(* PLC project cam_computation, Dassault Systèmes ControlBuild 2024x *)
(* stored: creationDateTime 2023-10-04T11:03:50-01:00 *)

(* This module simulates the behavior of a cam profile running module *)
FUNCTION_BLOCK motion_lib.cam_computation
  VAR_INPUT
    profileNr : DINT := 0;
    MasterPositionIn : REAL := 0.0;
  END_VAR
  VAR_INPUT
    nbPoints0 : INT := 0;
    MasterPoints0 : ARRAY[1..100] OF REAL := [100(0.0)];
    SlavePoints0 : ARRAY[1..100] OF REAL := [100(0.0)];
    pointer0 : DINT := 0;
  END_VAR
  VAR_INPUT
    nbPoints1 : INT := 0;
    MasterPoints1 : ARRAY[1..100] OF REAL := [100(0.0)];
    SlavePoints1 : ARRAY[1..100] OF REAL := [100(0.0)];
    pointer1 : DINT := 0;
  END_VAR
  VAR_INPUT
    nbPoints2 : INT := 0;
    MasterPoints2 : ARRAY[1..100] OF REAL := [100(0.0)];
    SlavePoints2 : ARRAY[1..100] OF REAL := [100(0.0)];
    pointer2 : DINT := 0;
  END_VAR
  VAR_INPUT
    nbPoints3 : INT := 0;
    MasterPoints3 : ARRAY[1..100] OF REAL := [100(0.0)];
    SlavePoints3 : ARRAY[1..100] OF REAL := [100(0.0)];
    pointer3 : DINT := 0;
  END_VAR
  VAR_OUTPUT
    slavePosition : REAL := 0.0;
    masterPosition : REAL := 0.0;
  END_VAR
  VAR
    i : INT := 0;
    modulo : REAL := 0.0;
    divider : INT := 0;
    faultProfileNr : BOOL := false;
    faultMasterPositionOOB : BOOL := false;
    faultLinComputation : BOOL := false;
    nbPoints : INT := 0;
    MasterPoints : ARRAY[1..100] OF REAL := [100(0.0)];
    SlavePoints : ARRAY[1..100] OF REAL := [100(0.0)];
    found : BOOL := false;
    index : INT := 0;
    linDenom : REAL := 0.0;
    linNum : REAL := 0.0;
    linA : REAL := 0.0;
    linB : REAL := 0.0;
  END_VAR
  VAR CONSTANT
    FACTOR : REAL := 1.0;
  END_VAR


ACTION C_source_code:
/* ----------------------------------------------------------------	*/
/* Type : Model of Operative Behaviour					*/
/* Category : motion_control						*/
/* Author : Dassault Systemes						*/
/* Update date : June 2021							*/
/* ----------------------------------------------------------------	*/
/* This module do the Slave cam computation from one Master position	*/
/* The profile table inputs are provided by the module cam_profile	*/
/* It's possible to switch in real time between 4 different profiles	*/
/* ----------------------------------------------------------------	*/


if (profileNr<0 || profileNr>3) {
	faultProfileNr = 1;
} else {
	faultProfileNr = 0;
	if (profileNr==0 && nbPoints0) {
		camTable = pointer0;
		nbPoints = nbPoints0;
		for (i=1; i< 100; i++) {
			MasterPoints(i) = camTable->master[i-1];
			SlavePoints(i) = camTable->slave[i-1];
		}
		modulo = camTable->master[nbPoints-1];
	} else {
		if (profileNr==1 && nbPoints1) {
			camTable = pointer1;
			nbPoints = nbPoints1;
			for (i=1; i< 100; i++) {
				MasterPoints(i) = camTable->master[i-1];
				SlavePoints(i) = camTable->slave[i-1];
			}
			modulo = camTable->master[nbPoints-1];
		} else {
			if (profileNr==2 && nbPoints2) {
				camTable = pointer2;
				nbPoints = nbPoints2;
				for (i=1; i< 100; i++) {
					MasterPoints(i) = camTable->master[i-1];
					SlavePoints(i) = camTable->slave[i-1];
				}
				modulo = camTable->master[nbPoints-1];
			} else {
				if (profileNr==3 && nbPoints3) {
					camTable = pointer3;
					nbPoints = nbPoints3;
					for (i=1; i< 100; i++) {
						MasterPoints(i) = camTable->master[i-1];
						SlavePoints(i) = camTable->slave[i-1];
					}
					modulo = camTable->master[nbPoints-1];
				}
			}
		}
	}
	if (nbPoints >= 2) {
		masterPosition = MasterPositionIn - divider * modulo;
		while (masterPosition > modulo) {
			divider += 1;
			masterPosition = MasterPositionIn - divider * modulo;
		}
		while (masterPosition < 0) {
			divider -= 1;
			masterPosition = MasterPositionIn - divider * modulo;
		}
		found = 0;
		for (i=1; i<= nbPoints - 1 && found == 0; i++) {
			if (camTable->master[i-1] <= masterPosition && masterPosition <= camTable->master[i]) {
				index = i;
				found = 1;
			} 
		}
		if (!found) {
			faultMasterPositionOOB = 1;
			if (masterPosition < camTable->master[0]) {
				slavePosition = camTable->slave[0] * FACTOR;
			} else {
				slavePosition = SlavePoints(nbPoints) * FACTOR;
			}
		} else {
			linDenom = camTable->master[index] - camTable->master[index-1];
			if (linDenom != 0.0) {
				faultLinComputation = 0;
				linNum = camTable->slave[index] - camTable->slave[index-1];
				linA = linNum / linDenom;
				linB = camTable->slave[index-1] - (linA * camTable->master[index-1]);
				slavePosition = FACTOR * (linA * masterPosition + linB);
			} else {
				faultLinComputation = 1;
			}
		}
	} else {
		slavePosition = 0;
	}
}
END_ACTION

ACTION C_header:
typedef struct camTableStruct
{  
	float master[7000];
	float slave[7000];
} camTableStruct;

camTableStruct *camTable;
END_ACTION
END_FUNCTION_BLOCK
